// Mitsubishi GX Works2 project: 0624(PLS,PLF)   PLC: Q02/Q02H

PROGRAM MAIN
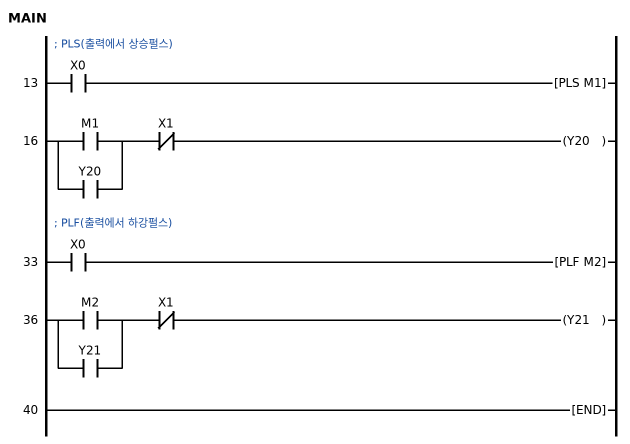
; PLS(출력에서 상승펄스)
13    LD      X0
      PLS     M1
16    LD      M1
      OR      Y20
      ANI     X1
      OUT     Y20
; PLF(출력에서 하강펄스)
33    LD      X0
      PLF     M2
36    LD      M2
      OR      Y21
      ANI     X1
      OUT     Y21
40    END
END_PROGRAM
